% RSLogix 500 project MOTOR_PR.RSS, saved by version 8.30.00.16 %
PROJECT "MOTOR_PR"    % processor: Bul.1763 MicroLogix 1100 Series B %

PROGRAM FILES
  LAD 2   2 rungs

DATA FILES
  O0 OUTPUT  4 elements
  I1 INPUT  6 elements
  S2 STATUS  66 elements
  B3 BINARY  1 elements
  T4 TIMER  1 elements
  C5 COUNTER  1 elements
  R6 CONTROL  1 elements
  N7 INTEGER  1 elements
  F8 FLOAT  1 elements

LADDER 2
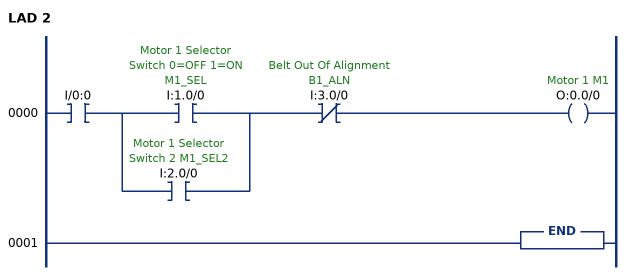
% Rung: 0 %  % edit flag set %
SOR XIC I/0:0 BST XIC I:1.0/0 NXB XIC I:2.0/0 BND XIO I:3.0/0 OTE O:0.0/0 EOR
%   I:1.0/0  M1_SEL  "Motor 1 Selector Switch 0=OFF 1=ON" %
%   I:2.0/0  M1_SEL2  "Motor 1 Selector Switch 2" %
%   I:3.0/0  B1_ALN  "Belt Out Of Alignment" %
%   O:0.0/0  M1  "Motor 1" %
% Rung: 1 %
SOR END EOR

OTHER DOCUMENTED ADDRESSES
  I:0  ES1  "Emergency Stop Push Buttton"
